// TwinCAT 3 PLC project VariablesPractice
// ProgramVersion: 3.1.4024.0
// libraries:
//   Tc2_Standard, * (Beckhoff Automation GmbH)
//   Tc2_System, * (Beckhoff Automation GmbH)
//   Tc3_Module, * (Beckhoff Automation GmbH)
// project tree:
//   / PlcTask.TcTTO
//   POUs/ FB_Car.TcPOU, FB_Motor.TcPOU, FB_TataNexon.TcPOU, I_Vehicle.TcIO, MAIN.TcPOU
// (motion and I/O tree: see PLC project functionblockpractice)
// real-time tasks:
//   TASK PlcTask: cycle T#10ms, priority 20, ADS port 350
//   TASK PlcTask2: cycle T#10ms, priority 22, ADS port 352
//   TASK PlcTask1: cycle T#10ms, priority 21, ADS port 351
//   TASK PlcTask3: cycle T#10ms, priority 23, ADS port 353
//   TASK PlcTask4: cycle T#10ms, priority 24, ADS port 354
//   TASK PlcTask5: cycle T#10ms, priority 25, ADS port 355
//   TASK PlcTask6: cycle T#10ms, priority 26, ADS port 356
//   TASK PlcTask7: cycle T#10ms, priority 27, ADS port 357

CONFIGURATION VariablesPractice
    RESOURCE PLC ON TwinCAT3
        TASK PlcTask(INTERVAL := T#10ms, PRIORITY := 27);
        PROGRAM MAIN WITH PlcTask : MAIN;
    END_RESOURCE
END_CONFIGURATION

// ---- POUs/I_Vehicle.TcIO
INTERFACE I_Vehicle

METHOD Drive : BOOL
VAR_INPUT
END_VAR
END_METHOD

END_INTERFACE

// ---- POUs/MAIN.TcPOU
PROGRAM MAIN
VAR
	nNum : DINT := 60000;
	fbMotor1 : FB_Motor ;
	fbMotor2 : FB_Motor ;
	
	fbTata : FB_TataNexon ;
	fbCar : POINTER TO FB_Car;
	
	iVehicle : I_Vehicle;
	pPoint1 : POINTER TO I_Vehicle;
	bRun: BOOL;
	num : INT;
	bCopyStart : BOOL;
END_VAR
VAR PERSISTENT
	num2 : INT := 323;
END_VAR
VAR CONSTANT
	num3 : INT := 34;
END_VAR

IF bRun THEN
	fbMotor1.Start();
	fbMotor1.Start();
	num := fbMotor1.nNum;
	fbMotor1.nNum := 433;
	bCopyStart := fbMotor1.bStart;
	bRun := FALSE;
END_IF
IF TRANS1 THEN
	//fbCar^.Running();
	fbTata();
END_IF
iVehicle := fbTata;
pPoint1 := ADR(iVehicle);

pPoint1^.Drive();

TRANSITION TRANS1:
TRANS1 := TRUE;
END_TRANSITION

END_PROGRAM

// ---- POUs/FB_Motor.TcPOU
FUNCTION_BLOCK FB_Motor

VAR_STAT
	{attribute 'hide'}
	nNum : INT;
END_VAR
VAR
	{attribute 'hide'}
	bStart : BOOL := TRUE;
END_VAR

IF TRANS_Check1 THEN
	nNum := 10;
END_IF

METHOD Start : BOOL
VAR_INPUT
END_VAR
nNum := nNum + 1;
END_METHOD

TRANSITION TRANS_Check1:
TRANS_Check1 := TRUE;
END_TRANSITION

END_FUNCTION_BLOCK

// ---- POUs/FB_TataNexon.TcPOU
FUNCTION_BLOCK FB_TataNexon EXTENDS FB_Car

VAR_INPUT
	nNum : INT;
END_VAR
VAR
	bStart : BOOL;
	bDriving : BOOL;
END_VAR

METHOD Drive : BOOL
VAR_INPUT
END_VAR
bDriving := TRUE;
END_METHOD

METHOD  Start : BOOL
VAR_INPUT
END_VAR
bStart := TRUE;
END_METHOD

END_FUNCTION_BLOCK

// ---- POUs/FB_Car.TcPOU
FUNCTION_BLOCK ABSTRACT FB_Car IMPLEMENTS I_Vehicle
VAR_INPUT
END_VAR
VAR_OUTPUT
END_VAR
VAR
END_VAR

METHOD Drive : BOOL
VAR_INPUT
END_VAR
END_METHOD

METHOD Running : BOOL
VAR_INPUT
END_VAR
END_METHOD

METHOD ABSTRACT Start : BOOL
VAR_INPUT
END_VAR
END_METHOD

END_FUNCTION_BLOCK
